PROGRAM motor_vfd_control_st
VAR PERSISTENT
END_VAR

END_PROGRAM

(* stored: Version 1.1.0.1, ProductVersion 3.1.4024.12
   POU motor_vfd_control_st: Id {a46dfc99-89d7-4ba2-a2c1-28118d28ec13}, SpecialFunc None *)
